FUNCTION_BLOCK DEV_CtrlValve EXTENDS FB_DeviceBase IMPLEMENTS ITF_ControlValve
VAR_INPUT
END_VAR
VAR_OUTPUT
END_VAR
VAR
END_VAR

{warning 'add property implementation'}
PROPERTY EmergencyStatus : BOOL
GET
END_GET
END_PROPERTY

{warning 'add property implementation'}
PROPERTY OperatingMode : BOOL
GET
END_GET
END_PROPERTY

{warning 'add property implementation'}
PROPERTY OutputValue : REAL
GET
END_GET
END_PROPERTY

{warning 'add method implementation '}
METHOD Reset : BOOL
END_METHOD

{warning 'add method implementation '}
METHOD SetMode : BOOL
END_METHOD

{warning 'add method implementation '}
METHOD SetValue : BOOL
END_METHOD

END_FUNCTION_BLOCK

(* stored: Version 1.1.0.1, ProductVersion 3.1.4024.12
   POU DEV_CtrlValve: Id {043053a6-7b48-43c8-bd59-f40d6b2e6cf6}, SpecialFunc None
   Property EmergencyStatus: Id {ba56147c-1df4-438b-9e8d-d96413157271}
   Get Get: Id {f44389a1-1a16-4e18-8a07-eb319156b66d}
   Property OperatingMode: Id {6155f774-466a-4b06-a07e-b1c3d9d1a1fb}
   Get Get: Id {1493a446-54ee-44f5-b87b-4cbe3887338d}
   Property OutputValue: Id {202d5ed9-938b-4e67-b830-87ca62464f61}
   Get Get: Id {db298ae9-eede-4b2e-b448-1a16b6fa8931}
   Method Reset: Id {ae730ef3-0d50-4721-b1b3-6c7c7496d3da}
   Method SetMode: Id {d4299c39-f6d2-4b87-8a2c-608b0523b815}
   Method SetValue: Id {74c20a76-b9ce-41ee-b396-fd85e0af7c41} *)
